PROGRAM MAIN
VAR
	byByte		AT %MB0	: ARRAY[0..1027] OF BYTE;
	i					: INT;
	moreBytes			: ARRAY[0..8192] OF BYTE;
	stInput				: ST_Packed;
	stOutput			: ST_Packed;
	stAlignedInput		: ST_Aligned;
	stAlignedOutput		: ST_Aligned;
	uAlignedInput		: U_AlignedStructs;
	uAlignedOutput		: U_AlignedStructs;
END_VAR

FOR i := 4 TO 1027 BY 1 DO
	byByte[i] := byByte[i] + 1;
END_FOR
stOutput := stInput;
stAlignedOutput := stAlignedInput;
uAlignedOutput.aAlignedStructs := uAlignedInput.aAlignedStructs;

END_PROGRAM

(* stored: Version 1.1.0.1, ProductVersion 3.1.4024.4
   POU MAIN: Id {f37b12b3-3b94-4389-b989-0323a722ff36}, SpecialFunc None *)
